// TwinCAT 3 PLC project Aufgabenserie_3
// ProgramVersion: 3.1.4022.3
// libraries:
//   Tc2_Standard, * (Beckhoff Automation GmbH)
//   Tc2_System, * (Beckhoff Automation GmbH)
//   Tc3_Module, * (Beckhoff Automation GmbH)
// project tree:
//   DUTs/ FSM_Deb.TcDUT, FSM_states.TcDUT
//   / GlobalTextList.TcGTLO (not stored), PlcTask.TcTTO, Visualisierungsmanager.TcVMO (not stored)
//   GVLs/ GVL_const.TcGVL (not stored), GVL_IO.TcGVL (not stored)
//   POUs/ fb_edgeDetector.TcPOU (not stored), MAIN.TcPOU
//   VISUs/ Visualization.TcVIS (not stored)
// real-time tasks:
//   TASK PlcTask: cycle T#10ms, priority 20, ADS port 350
// I/O:
//   DEVICE Gerät 1 (EtherCAT), AmsNetId 10.155.224.53.2.1
//     Klemme 1 (EK1200) [EK1200-5000 EtherCAT Netzteil (2A E-Bus)]
//       Klemme 2 (EL1004) [EL1004 4K. Dig. Eingang 24V, 3ms]
//       Klemme 3 (EL2004) [EL2004 4K. Dig. Ausgang 24V, 0.5A]
//       Klemme 4 (EL3004) [EL3004 4K.Ana. Eingang  +/-10V]
//       Klemme 5 (EL4034) [EL4034 4K. Ana. Ausgang +/-10V, 12bit]
//       Klemme 6 (EK1110) [EK1110 EtherCAT-Verlängerung]
//     Klemme 7 (EK1100) [EK1100 EtherCAT-Koppler (2A E-Bus)]
//       Klemme 8 (EL3004) [EL3004 4K.Ana. Eingang  +/-10V]
//       Klemme 9 (EL4032) [EL4032 2K. Ana. Ausgang +/-10V, 12bit]
//       Klemme 10 (EL9011) [EL9011 Endklemme]
//   DEVICE Gerät 2 (EtherCAT Automation Protocol) (disabled), AmsNetId 10.155.224.53.3.1
//   DEVICE Gerät 4 (EtherCAT Automation Protocol), AmsNetId 5.12.140.202.5.1
//   DEVICE Gerät 6 (EtherCAT), AmsNetId 5.12.140.202.7.1
//     Klemme 11 (EK1100) [EK1100 EtherCAT-Koppler (2A E-Bus)]
//       Klemme 12 (EL6900) [EL6900, TwinSAFE-PLC]
//       Klemme 13 (EL1904) [EL1904, 4 K. Safety Eingang 24V, TwinSAFE]
//         modules: Module 1 (FSOES)
//       Klemme 14 (EL2904) [EL2904, 4 K. Safety Ausgang 24V, 0.5A, TwinSAFE]
//         modules: Module 1 (FSOES), Module 2 (DO)
//       Klemme 5 (EL9011) [EL9011 Endklemme]
// variable links:
//   Aufgabenserie_3/Aufgabenserie_3 Instance <-> Device 1 (EtherCAT)/Term 1 (EK1200)/Term 2 (EL1004)
//     PlcTask Inputs/GVL_IO.b_blue_button <-> Channel 2/Input
//     PlcTask Inputs/GVL_IO.b_yellow_button <-> Channel 1/Input
//   Aufgabenserie_3/Aufgabenserie_3 Instance <-> Device 1 (EtherCAT)/Term 1 (EK1200)/Term 3 (EL2004)
//     PlcTask Outputs/GVL_IO.b_green_lamp <-> Channel 2/Output
//     PlcTask Outputs/GVL_IO.b_red_lamp <-> Channel 1/Output

CONFIGURATION Aufgabenserie_3
    RESOURCE PLC ON TwinCAT3
        TASK PlcTask(INTERVAL := T#10ms, PRIORITY := 20);
        PROGRAM MAIN WITH PlcTask : MAIN;
    END_RESOURCE
END_CONFIGURATION

// ---- DUTs/FSM_Deb.TcDUT
{attribute 'qualified_only'}
{attribute 'strict'}
TYPE FSM_Deb :
(
	deb_state_init := 0,
	deb_state_low,
	deb_state_rising,
	deb_state_high,
	deb_state_doble_activ,
	deb_state_falling
);
END_TYPE

// ---- DUTs/FSM_states.TcDUT
{attribute 'qualified_only'}
{attribute 'strict'}
TYPE FSM_states :
(
	state_init := 0,
	state_close,
	state_check,
	state_wrong,
	state_open,
	state_goChange,
	state_codChange,
	state_Res
);
END_TYPE

// ---- POUs/MAIN.TcPOU
PROGRAM MAIN
VAR
	st_current_state		:	FSM_states		:= FSM_states.state_init;
	
	fb_edgeDed_yellow		: 	fb_edgeDetector;
	fb_edgeDed_blue			:	fb_edgeDetector;
	
	b_array_code			:	ARRAY[0..3] OF BOOL		:=	[FALSE,TRUE,FALSE,TRUE];
	i_currentIndex			:	INT;
	t_correctCounter		:	TIME := T#0MS;
	
	i_wait_CodeChange		:	INT;
	
	
END_VAR

CASE st_current_state OF
	FSM_states.state_init:

		st_current_state	:=	FSM_states.state_close;
	FSM_states.state_close:
	
		GVL_IO.b_red_lamp	:=	FALSE;
		GVL_IO.b_green_lamp	:=	FALSE;
		i_currentIndex		:=	0;
		t_correctCounter	:=	T#0MS;
		i_wait_CodeChange	:=	0;
		
		st_current_state	:=	FSM_states.state_check;
			
	FSM_states.state_check:
		
		fb_edgeDed_blue(b_inputVal:=GVL_IO.b_blue_button);
		fb_edgeDed_yellow(b_inputVal:=GVL_IO.b_yellow_button);
		IF fb_edgeDed_blue.b_risingEdge THEN
			IF b_array_code[i_currentIndex]=FALSE THEN
				i_currentIndex		:=	i_currentIndex+1;
			ELSE
				st_current_state	:=	FSM_states.state_wrong;	
			END_IF
		ELSIF fb_edgeDed_yellow.b_risingEdge THEN
			IF b_array_code[i_currentIndex]=TRUE THEN
				i_currentIndex		:=	i_currentIndex+1;
			ELSE
				st_current_state	:=	FSM_states.state_wrong;	
			END_IF
		ELSIF fb_edgeDed_blue.b_doubleActivate THEN
			st_current_state	:=	FSM_states.state_Res;			
		END_IF
		
		IF i_currentIndex > 3 THEN
			st_current_state		:=	FSM_states.state_open;	
		END_IF
	FSM_states.state_Res:
		t_correctCounter	:=	t_correctCounter+GVL_const.T_CLOCK_CICLE;
		IF t_correctCounter=T#50MS THEN
			GVL_IO.b_green_lamp		:= NOT GVL_IO.b_green_lamp;
			GVL_IO.b_red_lamp		:= NOT GVL_IO.b_red_lamp;
		ELSIF t_correctCounter=T#100MS THEN
			GVL_IO.b_green_lamp		:= NOT GVL_IO.b_green_lamp;
			GVL_IO.b_red_lamp		:= NOT GVL_IO.b_red_lamp;
		ELSIF t_correctCounter=T#150MS THEN
			GVL_IO.b_green_lamp		:= NOT GVL_IO.b_green_lamp;
			GVL_IO.b_red_lamp		:= NOT GVL_IO.b_red_lamp;
		ELSIF t_correctCounter=T#200MS THEN
			GVL_IO.b_green_lamp		:= NOT GVL_IO.b_green_lamp;
			GVL_IO.b_red_lamp		:= NOT GVL_IO.b_red_lamp;
		ELSIF t_correctCounter=T#250MS THEN
			GVL_IO.b_green_lamp		:= NOT GVL_IO.b_green_lamp;
			GVL_IO.b_red_lamp		:= NOT GVL_IO.b_red_lamp;
		ELSIF t_correctCounter>T#300MS THEN
			st_current_state	:= FSM_states.state_init;
		END_IF
	
	FSM_states.state_wrong:
		
		IF t_correctCounter < GVL_const.T_LIGHT_DURATION THEN
			GVL_IO.b_red_lamp		:=	TRUE;
			t_correctCounter		:=	t_correctCounter + GVL_const.T_CLOCK_CICLE;
		ELSE
			st_current_state		:=	FSM_states.state_init;
		END_IF
	
	FSM_states.state_open:
		
		IF t_correctCounter < GVL_const.T_LIGHT_DURATION THEN
			GVL_IO.b_green_lamp		:=	TRUE;
			t_correctCounter		:=	t_correctCounter + GVL_const.T_CLOCK_CICLE;
		ELSE
			st_current_state		:=	FSM_states.state_init;
		END_IF
		
		
		IF GVL_IO.b_blue_button AND GVL_IO.b_yellow_button THEN
			st_current_state		:= FSM_states.state_goChange;
			i_currentIndex			:=0;
		END_IF
		
	FSM_states.state_goChange:
	
		fb_edgeDed_blue(b_inputVal			:=	GVL_IO.b_blue_button);
		fb_edgeDed_yellow(b_inputVal		:=	GVL_IO.b_yellow_button);
		
		IF fb_edgeDed_blue.b_fallingEdge OR fb_edgeDed_yellow.b_fallingEdge THEN
			i_wait_CodeChange				:=	i_wait_CodeChange+1;
		END_IF
		IF i_wait_CodeChange > 1 THEN
			st_current_state				:=	FSM_states.state_codChange;
		END_IF
		
		
	FSM_states.state_codChange:
		GVL_IO.b_green_lamp			:=	TRUE;
		GVL_IO.b_red_lamp			:=	TRUE;
		
		fb_edgeDed_blue(b_inputVal			:=GVL_IO.b_blue_button);
		fb_edgeDed_yellow(b_inputVal		:=GVL_IO.b_yellow_button);
		
		IF fb_edgeDed_blue.b_risingEdge THEN
			b_array_code[i_currentIndex]	:=	FALSE;
			i_currentIndex					:=	i_currentIndex+1;
		ELSIF fb_edgeDed_yellow.b_risingEdge THEN
			b_array_code[i_currentIndex]	:=	TRUE;
			i_currentIndex					:=	i_currentIndex+1;
		END_IF
		
		IF i_currentIndex > 3 THEN
			st_current_state				:=	FSM_states.state_init;
		END_IF
	
		
	
		
	
	
END_CASE

END_PROGRAM
